// TwinCAT 3 PLC project PLC_CRIX_MOT
// Title: lcls-plc-crix-motion
// Company: SLAC
// ProjectVersion: 2.5.0
// ProgramVersion: 3.1.4023.0
// libraries:
//   LCLS General, * (SLAC)
//   lcls-twincat-motion, * (SLAC)
//   PMPS, * (SLAC - LCLS)
//   Tc2_MC2, * (Beckhoff Automation GmbH)
//   Tc2_Standard, * (Beckhoff Automation GmbH)
//   Tc2_System, * (Beckhoff Automation GmbH)
//   Tc3_EventLogger, * (Beckhoff Automation GmbH)
//   Tc3_Module, * (Beckhoff Automation GmbH)
// project tree:
//   DUTs/Assemblies/ ENUM_DiagPaddle.TcDUT (not stored), ENUM_DPX.TcDUT (not stored), ENUM_DPY.TcDUT (not stored), ENUM_DPZ.TcDUT (not stored), E_DPaddle_States.TcDUT (not stored), ST_DiagPaddleOutputs.TcDUT (not stored)
//   Version/ Global_Version.TcGVL
//   DUTs/EPS/ ST_BFSAssemblyState.TcDUT (not stored), ST_EPSLimits.TcDUT (not stored), ST_Queue.TcDUT (not stored)
//   GVLs/ GVL.TcGVL, GVL_DiagnosticPaddle.TcGVL (not stored), GVL_FiberLite.TcGVL (not stored), GVL_Illumination.TcGVL (not stored), GVL_MotorEPS.TcGVL (not stored), GVL_PMPS.TcGVL (not stored), GVL_PointDetector.TcGVL (not stored), GVL_Questar.TcGVL (not stored), GVL_SampleDelivery.TcGVL (not stored), Main.TcGVL (not stored)
//   / PlcTask.TcTTO (not stored)
//   POUs/Assemblies/ FB_DPX.TcPOU (not stored), PRG_Beamblock.TcPOU (not stored), PRG_Camera.TcPOU (not stored), PRG_CryoPump.TcPOU (not stored), PRG_Cryopumps.TcPOU (not stored), PRG_CryoStat.TcPOU (not stored), PRG_DiagnosticPaddle.TcPOU (not stored), PRG_DiagnosticPaddleMotors.TcPOU (not stored), PRG_FiberLite.TcPOU (not stored), PRG_Illumination.TcPOU (not stored), PRG_InjectorMotors.TcPOU (not stored), PRG_PointDetectorMotors.TcPOU (not stored), PRG_ObjectivesMotors.TcPOU (not stored), PRG_QuestarMotors.TcPOU (not stored), PRG_RCC.TcPOU (not stored), PRG_RCI.TcPOU (not stored), PRG_VLS.TcPOU (not stored), PRG_SL2K2_SCATTER.TcPOU (not stored)
//   POUs/EPS/ FB_AdjacentStates.TcPOU (not stored), FB_AssemblyPositionStateManager.TcPOU (not stored), FB_BFS.TcPOU (not stored), FB_Queue.TcPOU (not stored), PRG_BFS.TcPOU (not stored), PRG_QueueTest.TcPOU (not stored), PRG_Test_AdjacentStates.TcPOU (not stored)
//   POUs/EPS/InjectorMotorEPSLimits/ FB_CheckEPS.TcPOU (not stored), F_InRange.TcPOU (not stored), FB_RestTimer.TcPOU (not stored), PRG_DPL_X_EPS.TcPOU (not stored), PRG_DPL_Y_EPS.TcPOU (not stored), PRG_DPL_Z_EPS.TcPOU, PRG_EPS.TcPOU, PRG_OBJ_X_EPS.TcPOU (not stored), PRG_RCC_Y_EPS.TcPOU (not stored), PRG_RCC_Z_EPS.TcPOU (not stored), PRG_SDS_RX_EPS.TcPOU (not stored), PRG_SDS_Y_EPS.TcPOU (not stored), PRG_SDS_ZENCODER_EPS.TcPOU (not stored)
//   POUs/ FB_RCI_Analog_Input.TcPOU (not stored), FB_RCI_Analog_Output.TcPOU (not stored), PRG_Main.TcPOU (not stored), PRG_PMPS.TcPOU (not stored)
//   POUs/temp/ FB_SLITS.TcPOU (not stored), FB_SLITS_POWER.TcPOU (not stored), FB_SLITS_SCATTER.TcPOU (not stored)

// ---- Version/Global_Version.TcGVL
{attribute 'TcGenerated'}
{attribute 'no-analysis'}
{attribute 'linkalways'}
// This function has been automatically generated from the project information.
VAR_GLOBAL CONSTANT
    {attribute 'const_non_replaced'}
    stLibVersion_lcls_plc_crix_motion : ST_LibVersion := (iMajor := 2, iMinor := 5, iBuild := 0, iRevision := 0, nFlags := 1, sVersion := '2.5.0');
END_VAR

// ---- GVLs/GVL.TcGVL
{attribute 'qualified_only'}
VAR_GLOBAL	
	xOverride		:	BOOL := FALSE; // Global override of motion safety settings.
END_VAR

// ---- POUs/EPS/InjectorMotorEPSLimits/PRG_DPL_Z_EPS.TcPOU
PROGRAM PRG_DPL_Z_EPS
VAR
    {attribute 'pytmc' := 'pv: CRIX:DPL:MMS:Z:EPS'}
    aDPL_Z_EPS 	    : ARRAY [1 .. 4] OF ST_EPSLimits;

    {attribute 'pytmc' := 'pv: CRIX:DPL:MMS:Z:EPS:OVRD_MODE'}
    bEPS_Override: BOOL := FALSE;
    {attribute 'pytmc' := 'pv: CRIX:DPL:MMS:Z:EPS:OVRD_COUNTDOWN'}
    tEPS_TimerCountDown : STRING := TIME_TO_STRING(T#0s);
    fbResetTimer : FB_RestTimer;

    bInit 		: BOOL := TRUE;
    bFullRange 	: BOOL;

    fbEPS		: FB_EPS;
    fbCheckEPS 	: FB_CheckEPS;
END_VAR

IF bInit THEN
    // Set Inital Values
    aDPL_Z_EPS[1].fBwd_Limits := -10;
    aDPL_Z_EPS[1].fFwd_Limits := 100;

    aDPL_Z_EPS[2].fBwd_Limits := 30;
    aDPL_Z_EPS[2].fFwd_Limits := 100;

    aDPL_Z_EPS[3].fBwd_Limits := 30;
    aDPL_Z_EPS[3].fFwd_Limits := 100;

    aDPL_Z_EPS[4].fBwd_Limits := 30;
    aDPL_Z_EPS[4].fFwd_Limits := 100;

    bInit := FALSE;
END_IF

fbEPS(eps:=aDPL_Z_EPS[2].stEPS);
fbEPS.setMessage('DPL X in [10, OBJ_X + 30]');
fbEPS.setBit(0, F_InRange(fDPL_X, 10, fOBJ_X + 30));

fbEPS(eps:=aDPL_Z_EPS[3].stEPS);
fbEPS.setMessage('RCC Y in [-34,10];RCC_Z in [-15,11]');
fbEPS.setBit(0, F_InRange(fRCC_Y, -34, 10));
fbEPS.setBit(1, F_InRange(fRCC_Z, -15, 11));

fbEPS(eps:=aDPL_Z_EPS[4].stEPS);
fbEPS.setMessage('RCC_Y in [-38,-34];RCC_Z in [-15,11];DPL_Y in [-1,40]');
fbEPS.setBit(0, F_InRange(fRCC_Y, -38, -34));
fbEPS.setBit(1, F_InRange(fRCC_Z, -15, 11));
fbEPS.setBit(2, F_InRange(fDPL_Y, -1, 40));

bFullRange := (NOT aDPL_Z_EPS[2].stEPS.bEPS_OK) AND (NOT aDPL_Z_EPS[3].stEPS.bEPS_OK) AND (NOT aDPL_Z_EPS[4].stEPS.bEPS_OK);

fbEPS(eps:=aDPL_Z_EPS[1].stEPS);
fbEPS.setMessage('Full Range');
fbEPS.setBit(0, bFullRange);

fbResetTimer(bInput:=bEPS_Override, tElapseTime:=tEPS_OVRD_RESET_TIME, tCountDown:=tEPS_TimerCountDown);
fbCheckEPS(stMotor:=M3, fPosition:=fDPL_Z, aEPSLimits:= aDPL_Z_EPS, stForwardMotorEPS:=M3.stEPSForwardEnable, stBackwardMotorEPS:= M3.stEPSBackwardEnable, bEPS_Override:=bEPS_Override);

END_PROGRAM

// ---- POUs/EPS/InjectorMotorEPSLimits/PRG_EPS.TcPOU
PROGRAM PRG_EPS
VAR
END_VAR

// Update Motor Positions before Using them in EPS Checks
fDPL_X  	:= M1.stAxisStatus.fActPosition;

fSDS_RX 	:= M19.stAxisStatus.fActPosition;
fSDS_Y      := M17.stAxisStatus.fActPosition;
fSDS_Z_ENC  := M36.stAxisStatus.fActPosition;

fDPL_Z 		:= M3.stAxisStatus.fActPosition;
fDPL_Y 		:= M2.stAxisStatus.fActPosition;

fRCC_Z 		:= M39.stAxisStatus.fActPosition;
fRCC_Y 		:= M38.stAxisStatus.fActPosition;

fOBJ_X		:= M4.stAxisStatus.fActPosition;

PRG_SDS_Y_EPS();
PRG_SDS_RX_EPS();
PRG_SDS_ZENCODER_EPS();

PRG_DPL_X_EPS();
PRG_DPL_Y_EPS();
PRG_DPL_Z_EPS();

PRG_RCC_Y_EPS();
PRG_RCC_Z_EPS();

PRG_OBJ_X();

END_PROGRAM
